(* IEC 61131-3 sources: repolevel_ST_code_completion/output/0122完整版本_无planner目前sota/repoeval_electronic_cam_motion/readful_result_no_provide, 4 files *)

(* ---- F_AxisStatusToString.st ---- *)
IF fbReadStatus.Errorstop THEN
	F_AxisStatusToString := 'Errorstop';
	RETURN;
END_IF

IF fbReadStatus.Disabled THEN
	F_AxisStatusToString := 'Disabled';
	RETURN;
END_IF

IF fbReadStatus.Homing THEN
	F_AxisStatusToString := 'Homing';
	RETURN;
END_IF

IF fbReadStatus.Stopping THEN
	F_AxisStatusToString := 'Stopping';
	RETURN;
END_IF

IF fbReadStatus.SynchronizedMotion THEN
	F_AxisStatusToString := 'SynchronizedMotion';
	RETURN;
END_IF

IF fbReadStatus.ContinuousMotion THEN
	F_AxisStatusToString := 'ContinuousMotion';
	RETURN;
END_IF

IF fbReadStatus.Standstill THEN
	F_AxisStatusToString := 'Standstill';
	RETURN;
END_IF

F_AxisStatusToString := 'Unknown';
RETURN;
END_FUNCTION

(* ---- FB_DualAxisPower.st ---- *)
VAR
	fbPower1		:	MC_Power;			//轴1电源控制
	fbPower2		:	MC_Power;			//轴2电源控制
	bAxis1Error		:	BOOL;				//轴1错误标志
	bAxis2Error		:	BOOL;				//轴2错误标志
END_VAR

fbPower1(
	Axis := Axis1,
	Enable := TRUE,
	bDriveStart := bPowerOn,
	bRegulatorOn := bPowerOn
);

fbPower2(
	Axis := Axis2,
	Enable := TRUE,
	bDriveStart := bPowerOn,
	bRegulatorOn := bPowerOn
);

bAxis1Ready := fbPower1.Status = MC_POWER_STATUS_READY;
bAxis2Ready := fbPower2.Status = MC_POWER_STATUS_READY;

bAxis1Error := fbPower1.Error;
bAxis2Error := fbPower2.Error;

bError := bAxis1Error OR bAxis2Error;
bPowerDone := bAxis1Ready AND bAxis2Ready AND NOT bError;
END_FUNCTION_BLOCK

(* ---- FB_DualAxisReset.st ---- *)
VAR
	fbReset1		:	MC_Reset;			//轴1复位
	fbReset2		:	MC_Reset;			//轴2复位
	fbReadStatus1	:	MC_ReadStatus;		//轴1状态读取
	fbReadStatus2	:	MC_ReadStatus;		//轴2状态读取
	bError1			:	BOOL;				//轴1错误标志
	bError2			:	BOOL;				//轴2错误标志
	nState			:	UDINT;				//状态机
END_VAR

CASE nState OF
	0: (* 空闲状态 *)
		bDone := FALSE;
		bBusy := FALSE;
		bError := FALSE;

		IF bExecute THEN
			// 初始化
			fbReset1(Axis := Axis1, Execute := FALSE);
			fbReset2(Axis := Axis2, Execute := FALSE);
			fbReadStatus1(Axis := Axis1);
			fbReadStatus2(Axis := Axis2);
			nState := 1;
		END_IF;

	1: (* 检查轴状态 *)
		fbReadStatus1(Axis := Axis1);
		fbReadStatus2(Axis := Axis2);

		bError1 := fbReadStatus1.Error;
		bError2 := fbReadStatus2.Error;

		IF bError1 OR bError2 THEN
			bError := TRUE;
			nState := 0;
		ELSE
			nState := 2;
		END_IF;

	2: (* 执行复位 *)
		bBusy := TRUE;

		fbReset1(Axis := Axis1, Execute := TRUE);
		fbReset2(Axis := Axis2, Execute := TRUE);

		IF fbReset1.Done AND fbReset2.Done THEN
			bDone := TRUE;
			bBusy := FALSE;
			nState := 0;
		END_IF;

		IF fbReset1.Error OR fbReset2.Error THEN
			bError := TRUE;
			bBusy := FALSE;
			nState := 0;
		END_IF;

END_CASE;
END_FUNCTION_BLOCK

(* ---- ResetAxis.st ---- *)
VAR
	fbReset1	:	MC_Reset;
	fbReset2	:	MC_Reset;

	fbReadAxisError1	:	MC_ReadAxisError;
	fbReadAxisError2	:	MC_ReadAxisError;

	fbReadStatus1	:	MC_ReadStatus;
	fbReadStatus2	:	MC_ReadStatus;

	fbExecTrig	:	R_TRIG;
	nState 	:	BYTE;

	bErrorX	:	BOOL;
	bErrorY	:	BOOL;

END_VAR

VAR_OUTPUT
	Done	:	BOOL;
END_VAR

fbExecTrig(CLK := bExec);

CASE nState OF
	0:
		IF fbExecTrig.Q THEN
			nState := 1;
			Done := FALSE;
		END_IF
	1:
		fbReadAxisError1(Execute := TRUE);
		fbReadAxisError2(Execute := TRUE);

		bErrorX := fbReadAxisError1.Error;
		bErrorY := fbReadAxisError2.Error;

		IF NOT bErrorX AND NOT bErrorY THEN
			nState := 3;
		ELSE
			nState := 2;
		END_IF
	2:
		fbReset1(Execute := bErrorX);
		fbReset2(Execute := bErrorY);

		IF fbReset1.Done AND fbReset2.Done THEN
			nState := 3;
		END_IF
	3:
		fbReadStatus1(Execute := TRUE);
		fbReadStatus2(Execute := TRUE);

		IF fbReadStatus1.Error OR fbReadStatus2.Error THEN
			nState := 2;
		ELSE
			Done := TRUE;
			nState := 0;
		END_IF
END_CASE;
END_FUNCTION_BLOCK
